{attribute addProperty BoxType "EL3423-0000-0020"}
{attribute addProperty Id "Apparent_EnergyAT %I*LINT648"}
{attribute addProperty CRC "3706737417"}
{attribute addProperty SizeInBites "64"}
{attribute addProperty SizeInBytes "8"}
TYPE Total_Apparent_Reduced_DCF05309 :
STRUCT
	{attribute addProperty Name "Apparent_Energy"}
	Apparent_Energy AT %I* : LINT;
END_STRUCT
END_TYPE

(* stored: Version 1.2.0.0, ProductVersion 3.1.4024.9
   DUT Total_Apparent_Reduced_DCF05309: Id {68f98183-f7ca-4f0a-92e7-4038439bf9a1} *)
